FUNCTION_BLOCK overcurrentV2 (* Basic Function Block Type *)
  (* Standard: 61499-2 *)
  (* Version 0.0, 21/03/2016, Chen-Wei, nxtControl GmbH, Template *)
  PACKAGE Main;
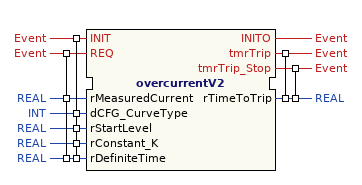
  EVENT_INPUT
    INIT WITH dCFG_CurveType, rStartLevel, rConstant_K, rDefiniteTime; (* Initialization Request *)
    REQ WITH rMeasuredCurrent, rDefiniteTime; (* Normal Execution Request *)
  END_EVENT
  EVENT_OUTPUT
    INITO; (* Initialization Confirm *)
    tmrTrip WITH rTimeToTrip; (* Execution Confirmation *)
    tmrTrip_Stop WITH rTimeToTrip;
  END_EVENT
  VAR_INPUT
    rMeasuredCurrent : REAL; (* Input event qualifier *)
    dCFG_CurveType : INT;
    rStartLevel : REAL;
    rConstant_K : REAL;
    rDefiniteTime : REAL;
  END_VAR
  VAR_OUTPUT
    rTimeToTrip : REAL;
  END_VAR
  VAR
    mStart : BOOL;
    rTimeToTripInternal : REAL;
    INT_dCFG_CurveType : INT;
    ans1 : REAL;
    ans2 : REAL;
    ans3 : REAL;
    veryLargeNumber : REAL := 9999999;
    TimerStarted : BOOL;
  END_VAR
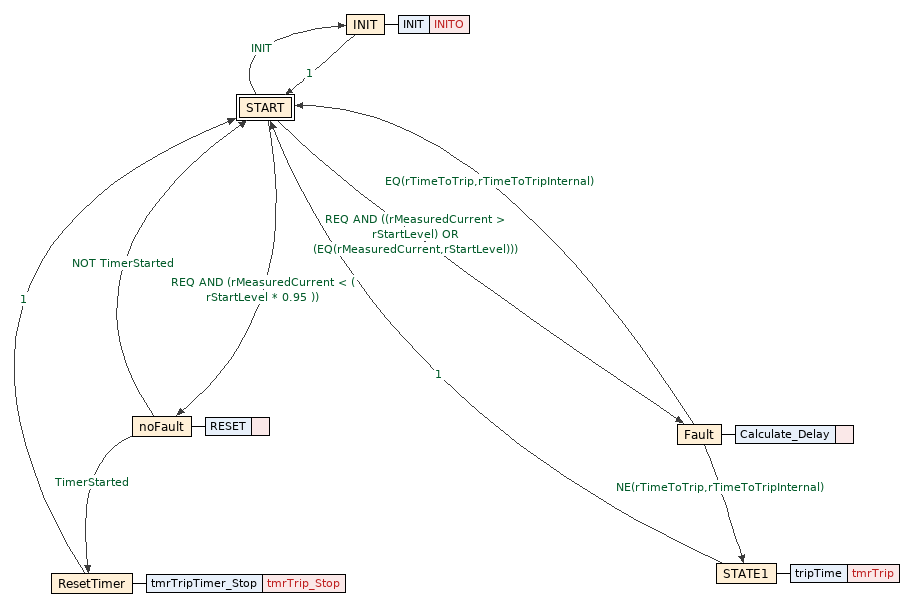
  EC_STATES
    START; (* Initial State *)
    INIT : INIT -> INITO; (* Initialization *)
    noFault : RESET;
    Fault : Calculate_Delay;
    ResetTimer : tmrTripTimer_Stop -> tmrTrip_Stop;
    STATE1 : tripTime -> tmrTrip;
  END_STATES
  EC_TRANSITIONS
    START TO INIT := INIT;
    INIT TO START := 1;
    START TO Fault := REQ AND ((rMeasuredCurrent > rStartLevel) OR (EQ(rMeasuredCurrent,rStartLevel)));
    START TO noFault := REQ AND (rMeasuredCurrent < ( rStartLevel * 0.95 ));
    Fault TO START := EQ(rTimeToTrip,rTimeToTripInternal);
    noFault TO ResetTimer := TimerStarted;
    ResetTimer TO START := 1;
    noFault TO START := NOT TimerStarted;
    Fault TO STATE1 := NE(rTimeToTrip,rTimeToTripInternal);
    STATE1 TO START := 1;
  END_TRANSITIONS
  ALGORITHM INIT IN ST: (* Initialization algorithm *)
INIT := 0;
mStart := FALSE;
TimerStarted := FALSE;


INT_dCFG_CurveType := dCFG_CurveType;


;
  END_ALGORITHM
  ALGORITHM RESET IN ST:
mStart := FALSE;
rTimeToTripInternal := 0.0;
;
  END_ALGORITHM
  ALGORITHM Calculate_Delay IN ST: (* Version:      2.01 2016-05-23 First Revision Curvtype: (dCFG_CurveType) 0 : Definite time 1: IEC Normal Inverse 2: IEC Very Inverse 3: IEC Extremely Inverse 4: RI Curve *)
(*
VAR
	ans1:REAL;
	ans2:REAL;
	ans3:REAL;
	veryLargeNumber:REAL:= 9999999;
END_VAR;*)

mStart := TRUE;

//IF mStart THEN
	(* Calculate time to trip *)
	CASE INT_dCFG_CurveType OF
		1: (* IEC Normal Inverse *)

  		IF (rStartLevel = 0.0) THEN
  			ans1 := EXPT(veryLargeNumber, 0.02);
  		ELSE
  			ans1 := EXPT((rMeasuredCurrent/rStartLevel) , 0.02);
  		END_IF;

  		IF ((ans1 - 1.0) = 0.0) THEN
  			ans2 := veryLargeNumber;
  		ELSE
  			ans2 := 0.14/(ans1 - 1.0);
  		END_IF;
  		rTimeToTripInternal := rConstant_K*ans2;

		2: (* IEC Very Inverse *)

  		IF (rStartLevel = 0.0) THEN
  			ans1 := veryLargeNumber - 1.0;
  		ELSE
  			ans1 := (rMeasuredCurrent/rStartLevel) - 1.0;
  		END_IF;

  		IF (ans1 = 0.0) THEN
  			ans2 := veryLargeNumber;
  		ELSE
  			ans2 := 13.5/ans1;
  		END_IF;
  		rTimeToTripInternal := rConstant_K*ans2;

		3: (* IEC Extremely Inverse *)

  		IF (rStartLevel = 0.0) THEN
  			ans1 := EXPT(veryLargeNumber, 2.0);
  		ELSE
  			ans1 := EXPT((rMeasuredCurrent/rStartLevel) , 2.0);
  		END_IF;

  		IF ((ans1 - 1.0) = 0.0) THEN
  			ans2 := veryLargeNumber;
  		ELSE
  			ans2 := 80.0/(ans1 - 1.0);
  		END_IF;
  		rTimeToTripInternal := rConstant_K*ans2;

		4: (* RI Curve *)

  		IF (rStartLevel = 0.0) THEN
  			ans1 := veryLargeNumber;
  		ELSE
  			ans1 := rMeasuredCurrent/rStartLevel;
  		END_IF;

  		IF (ans1 = 0.0) THEN
  			ans2 := veryLargeNumber;
  		ELSE
  			ans2 := 0.339-(0.236/ans1);
  		END_IF;

  		IF (ans2 = 0.0) THEN
  			ans3 := veryLargeNumber;
  		ELSE
  			ans3 := (1.0/ans2);
  		END_IF;
  		rTimeToTripInternal := rConstant_K*ans3;

		0: (* Definite Time *)
		  rTimeToTripInternal := rDefiniteTime;

	ELSE
		(* Definite Time *)
		rTimeToTripInternal := rDefiniteTime;
	END_CASE;
//END_IF;

//rTimeToTrip := rTimeToTripInternal;
//TimerStarted := TRUE;

//INT_dCFG_CurveType := dCFG_CurveType;

;
  END_ALGORITHM
  ALGORITHM tmrTripTimer_Stop IN ST:
rTimeToTrip := rTimeToTripInternal;
TimerStarted := FALSE;
;
  END_ALGORITHM
  ALGORITHM tripTime IN ST:
;
rTimeToTrip := rTimeToTripInternal;
TimerStarted := TRUE;
  END_ALGORITHM
END_FUNCTION_BLOCK
